# EPICS StreamDevice protocol: default.proto
Terminator = LF;

getBoolParam { out "R:\$1:"; in "R:\$1:%{False|True}"; }

setBoolParam { out "W:\$1:%s"; }

getAnalogParam { out "R:\$1:"; in "R:\$1:%f"; }

setAnalogParam { out "W:\$1:%f"; }

getStrParam { out "R:\$1:"; in "R:\$1:%s"; }

setStrParam { out "W:\$1:%s"; }
